PROGRAM Floor2
VAR
	floorTwoLamp : BOOL := FALSE;
END_VAR

END_PROGRAM

(* stored: Version 1.1.0.1, ProductVersion 3.1.4024.12
   POU Floor2: Id {1b66c6d5-e132-4dd6-bb1d-63572541cf58}, SpecialFunc None *)
